TYPE
    ST_IRC5_Command : STRUCT
        Extend  : BOOL;
        Retract : BOOL;
    END_STRUCT
END_TYPE

(* stored: Version 1.1.0.1
   DUT ST_IRC5_Command: Id {33d5f418-3572-4f11-a2ed-17b32de7ed39} *)
